// TIA Portal V17 export
// export: Created 2025-03-07T09:23:56.1617823Z, ExportSetting WithDefaults, DisplayName Totally Integrated Automation Portal, DisplayVersion V17 Update 8, DisplayName TIA Portal Openness, DisplayVersion V17 Update 8, DisplayName TIA Portal Version Control Interface, DisplayVersion V17, DisplayName SINAMICS Startdrive Advanced, DisplayVersion V17 SP2, DisplayName SINAMICS Startdrive G110M, G120, G120C, G120D, G120P, G115D, DisplayVersion V17 SP2, DisplayName SINAMICS Startdrive G130, G150, S120, S150, SINAMICS MV, S210, DisplayVersion V17 SP2, DisplayName STEP 7 Professional, DisplayVersion V17 Update 8, DisplayName SINUMERIK ONE STEP 7 Toolbox, DisplayVersion V17 Update 12, DisplayName SINUMERIK 840D sl STEP 7 Toolbox, DisplayVersion V17 Update 12, DisplayName STEP 7 Safety, DisplayVersion V17 Update 6, DisplayName WinCC Advanced, DisplayVersion V17 Update 8
FUNCTION "FC21200_POWDER_FLOW_SENSOR_MEDICOAT" : Void   // FC21200, LAD
{ S7_Optimized_Access := 'TRUE' }
VERSION : 0.1
// stored: AutoNumber false, IsIECCheckEnabled false, SetENOAutomatically false, UDAEnableTagReadback false
BEGIN

REGION Network 1: /////_UNIT_01_/////
END_REGION

REGION Network 2: OERLIKON 1 LINE 1 OUTPUT MEDICOAT
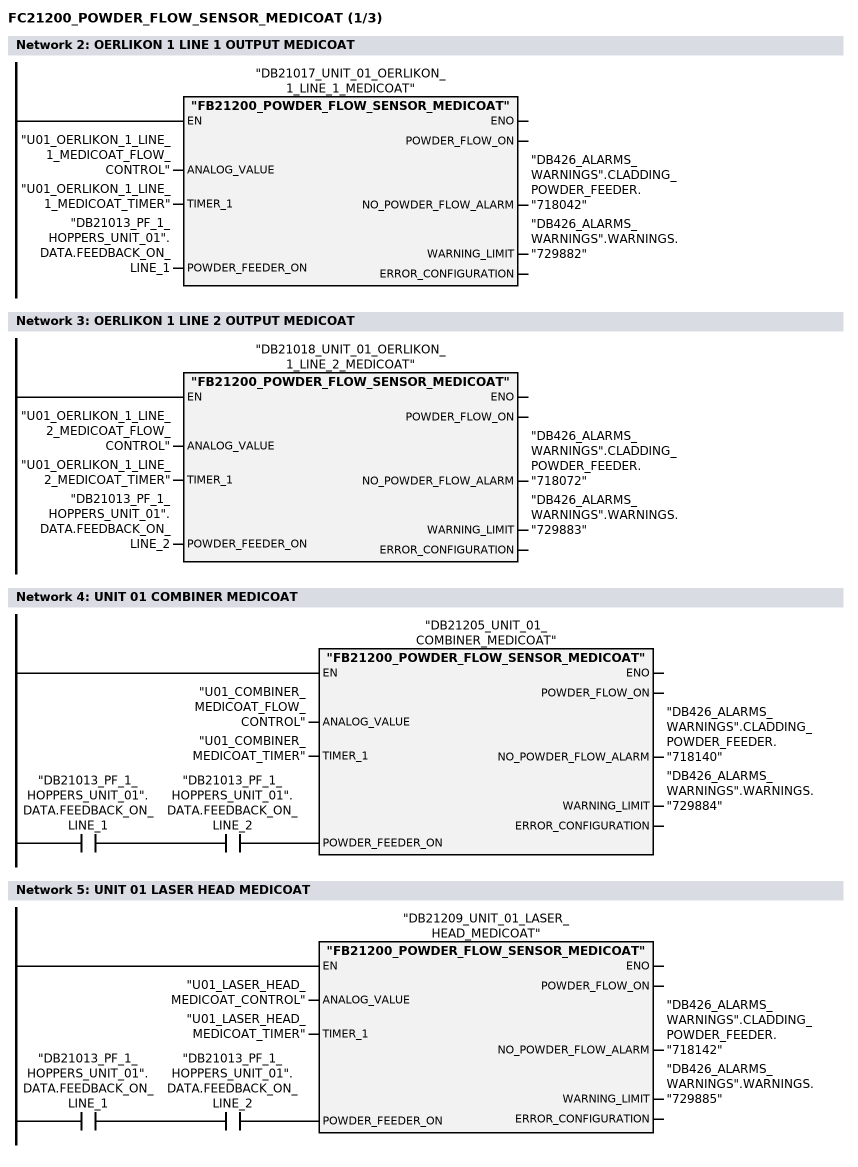
   RUNG wire#powerrail
      "DB21017_UNIT_01_OERLIKON_1_LINE_1_MEDICOAT"(ANALOG_VALUE := "U01_OERLIKON_1_LINE_1_MEDICOAT_FLOW_CONTROL", TIMER_1 := "U01_OERLIKON_1_LINE_1_MEDICOAT_TIMER", POWDER_FEEDER_ON := "DB21013_PF_1_HOPPERS_UNIT_01".DATA.FEEDBACK_ON_LINE_1, POWDER_FLOW_ON =>, NO_POWDER_FLOW_ALARM => "DB426_ALARMS_WARNINGS".CLADDING_POWDER_FEEDER."718042", WARNING_LIMIT => "DB426_ALARMS_WARNINGS".WARNINGS."729882", ERROR_CONFIGURATION =>)
   END_RUNG
   // the same network as SCL:
   "DB21017_UNIT_01_OERLIKON_1_LINE_1_MEDICOAT"(ANALOG_VALUE := "U01_OERLIKON_1_LINE_1_MEDICOAT_FLOW_CONTROL",   // "FB21200_POWDER_FLOW_SENSOR_MEDICOAT"
                           TIMER_1 := "U01_OERLIKON_1_LINE_1_MEDICOAT_TIMER",
                           POWDER_FEEDER_ON := "DB21013_PF_1_HOPPERS_UNIT_01".DATA.FEEDBACK_ON_LINE_1,
                           NO_POWDER_FLOW_ALARM => "DB426_ALARMS_WARNINGS".CLADDING_POWDER_FEEDER."718042",
                           WARNING_LIMIT => "DB426_ALARMS_WARNINGS".WARNINGS."729882");
END_REGION

REGION Network 3: OERLIKON 1 LINE 2 OUTPUT MEDICOAT
   RUNG wire#powerrail
      "DB21018_UNIT_01_OERLIKON_1_LINE_2_MEDICOAT"(ANALOG_VALUE := "U01_OERLIKON_1_LINE_2_MEDICOAT_FLOW_CONTROL", TIMER_1 := "U01_OERLIKON_1_LINE_2_MEDICOAT_TIMER", POWDER_FEEDER_ON := "DB21013_PF_1_HOPPERS_UNIT_01".DATA.FEEDBACK_ON_LINE_2, POWDER_FLOW_ON =>, NO_POWDER_FLOW_ALARM => "DB426_ALARMS_WARNINGS".CLADDING_POWDER_FEEDER."718072", WARNING_LIMIT => "DB426_ALARMS_WARNINGS".WARNINGS."729883", ERROR_CONFIGURATION =>)
   END_RUNG
   // the same network as SCL:
   "DB21018_UNIT_01_OERLIKON_1_LINE_2_MEDICOAT"(ANALOG_VALUE := "U01_OERLIKON_1_LINE_2_MEDICOAT_FLOW_CONTROL",   // "FB21200_POWDER_FLOW_SENSOR_MEDICOAT"
                           TIMER_1 := "U01_OERLIKON_1_LINE_2_MEDICOAT_TIMER",
                           POWDER_FEEDER_ON := "DB21013_PF_1_HOPPERS_UNIT_01".DATA.FEEDBACK_ON_LINE_2,
                           NO_POWDER_FLOW_ALARM => "DB426_ALARMS_WARNINGS".CLADDING_POWDER_FEEDER."718072",
                           WARNING_LIMIT => "DB426_ALARMS_WARNINGS".WARNINGS."729883");
END_REGION

REGION Network 4: UNIT 01 COMBINER MEDICOAT
   RUNG wire#powerrail
      "DB21205_UNIT_01_COMBINER_MEDICOAT"(POWDER_FEEDER_ON := wire#w1, ANALOG_VALUE := "U01_COMBINER_MEDICOAT_FLOW_CONTROL", TIMER_1 := "U01_COMBINER_MEDICOAT_TIMER", POWDER_FLOW_ON =>, NO_POWDER_FLOW_ALARM => "DB426_ALARMS_WARNINGS".CLADDING_POWDER_FEEDER."718140", WARNING_LIMIT => "DB426_ALARMS_WARNINGS".WARNINGS."729884", ERROR_CONFIGURATION =>)
   END_RUNG
   RUNG wire#powerrail
      Contact( "DB21013_PF_1_HOPPERS_UNIT_01".DATA.FEEDBACK_ON_LINE_1 )
      Contact( "DB21013_PF_1_HOPPERS_UNIT_01".DATA.FEEDBACK_ON_LINE_2 )
   END_RUNG wire#w1
   // the same network as SCL:
   "DB21205_UNIT_01_COMBINER_MEDICOAT"(ANALOG_VALUE := "U01_COMBINER_MEDICOAT_FLOW_CONTROL",   // "FB21200_POWDER_FLOW_SENSOR_MEDICOAT"
                           TIMER_1 := "U01_COMBINER_MEDICOAT_TIMER",
                           POWDER_FEEDER_ON := "DB21013_PF_1_HOPPERS_UNIT_01".DATA.FEEDBACK_ON_LINE_1 AND "DB21013_PF_1_HOPPERS_UNIT_01".DATA.FEEDBACK_ON_LINE_2,
                           NO_POWDER_FLOW_ALARM => "DB426_ALARMS_WARNINGS".CLADDING_POWDER_FEEDER."718140",
                           WARNING_LIMIT => "DB426_ALARMS_WARNINGS".WARNINGS."729884");
END_REGION

REGION Network 5: UNIT 01 LASER HEAD MEDICOAT
   RUNG wire#powerrail
      "DB21209_UNIT_01_LASER_HEAD_MEDICOAT"(POWDER_FEEDER_ON := wire#w1, ANALOG_VALUE := "U01_LASER_HEAD_MEDICOAT_CONTROL", TIMER_1 := "U01_LASER_HEAD_MEDICOAT_TIMER", POWDER_FLOW_ON =>, NO_POWDER_FLOW_ALARM => "DB426_ALARMS_WARNINGS".CLADDING_POWDER_FEEDER."718142", WARNING_LIMIT => "DB426_ALARMS_WARNINGS".WARNINGS."729885", ERROR_CONFIGURATION =>)
   END_RUNG
   RUNG wire#powerrail
      Contact( "DB21013_PF_1_HOPPERS_UNIT_01".DATA.FEEDBACK_ON_LINE_1 )
      Contact( "DB21013_PF_1_HOPPERS_UNIT_01".DATA.FEEDBACK_ON_LINE_2 )
   END_RUNG wire#w1
   // the same network as SCL:
   "DB21209_UNIT_01_LASER_HEAD_MEDICOAT"(ANALOG_VALUE := "U01_LASER_HEAD_MEDICOAT_CONTROL",   // "FB21200_POWDER_FLOW_SENSOR_MEDICOAT"
                           TIMER_1 := "U01_LASER_HEAD_MEDICOAT_TIMER",
                           POWDER_FEEDER_ON := "DB21013_PF_1_HOPPERS_UNIT_01".DATA.FEEDBACK_ON_LINE_1 AND "DB21013_PF_1_HOPPERS_UNIT_01".DATA.FEEDBACK_ON_LINE_2,
                           NO_POWDER_FLOW_ALARM => "DB426_ALARMS_WARNINGS".CLADDING_POWDER_FEEDER."718142",
                           WARNING_LIMIT => "DB426_ALARMS_WARNINGS".WARNINGS."729885");
END_REGION

REGION Network 6: /////_UNIT_02_/////
END_REGION

REGION Network 7: UNIT 02 OERLIKON 1 LINE 1 OUTPUT MEDICOAT
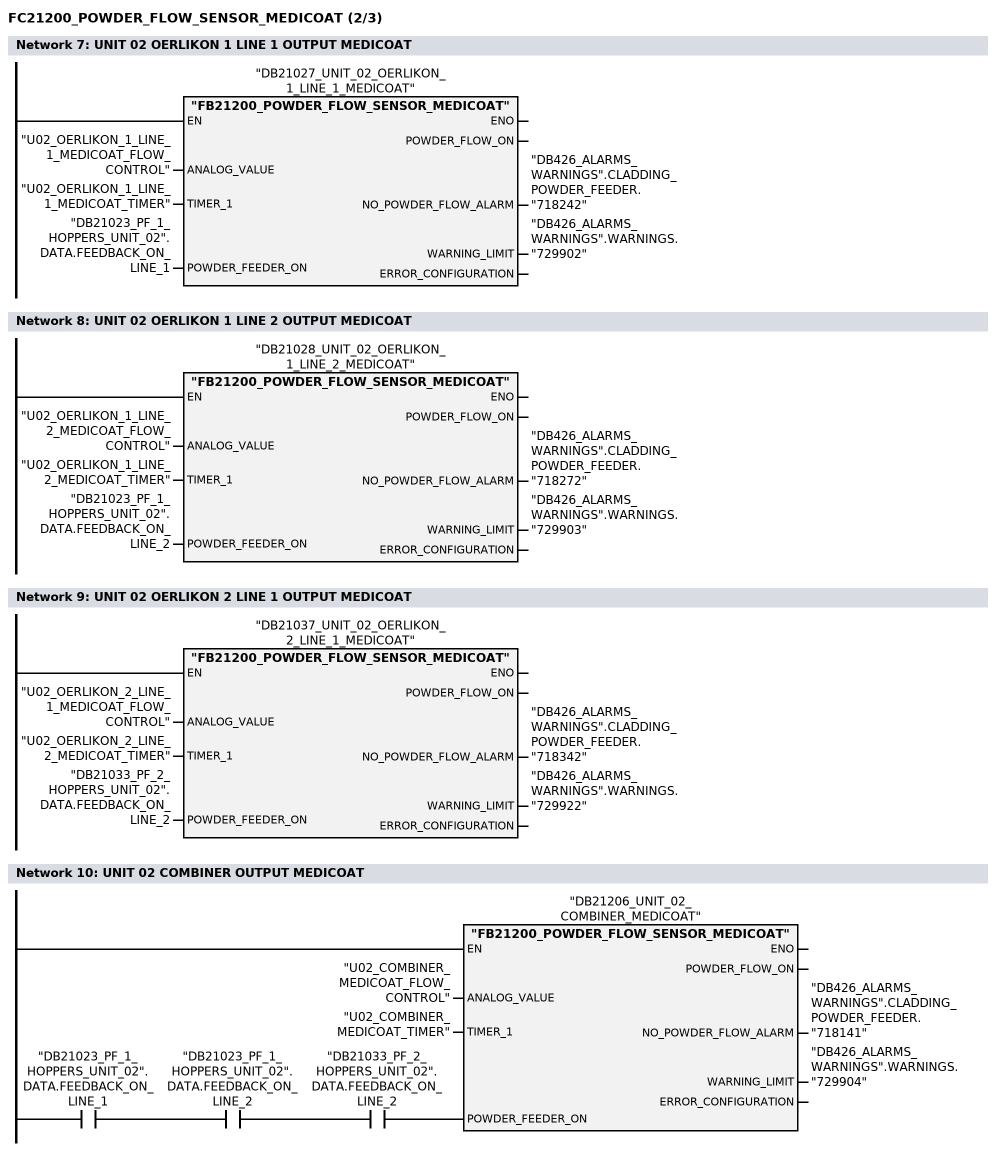
   RUNG wire#powerrail
      "DB21027_UNIT_02_OERLIKON_1_LINE_1_MEDICOAT"(ANALOG_VALUE := "U02_OERLIKON_1_LINE_1_MEDICOAT_FLOW_CONTROL", TIMER_1 := "U02_OERLIKON_1_LINE_1_MEDICOAT_TIMER", POWDER_FEEDER_ON := "DB21023_PF_1_HOPPERS_UNIT_02".DATA.FEEDBACK_ON_LINE_1, POWDER_FLOW_ON =>, NO_POWDER_FLOW_ALARM => "DB426_ALARMS_WARNINGS".CLADDING_POWDER_FEEDER."718242", WARNING_LIMIT => "DB426_ALARMS_WARNINGS".WARNINGS."729902", ERROR_CONFIGURATION =>)
   END_RUNG
   // the same network as SCL:
   "DB21027_UNIT_02_OERLIKON_1_LINE_1_MEDICOAT"(ANALOG_VALUE := "U02_OERLIKON_1_LINE_1_MEDICOAT_FLOW_CONTROL",   // "FB21200_POWDER_FLOW_SENSOR_MEDICOAT"
                           TIMER_1 := "U02_OERLIKON_1_LINE_1_MEDICOAT_TIMER",
                           POWDER_FEEDER_ON := "DB21023_PF_1_HOPPERS_UNIT_02".DATA.FEEDBACK_ON_LINE_1,
                           NO_POWDER_FLOW_ALARM => "DB426_ALARMS_WARNINGS".CLADDING_POWDER_FEEDER."718242",
                           WARNING_LIMIT => "DB426_ALARMS_WARNINGS".WARNINGS."729902");
END_REGION

REGION Network 8: UNIT 02 OERLIKON 1 LINE 2 OUTPUT MEDICOAT
   RUNG wire#powerrail
      "DB21028_UNIT_02_OERLIKON_1_LINE_2_MEDICOAT"(ANALOG_VALUE := "U02_OERLIKON_1_LINE_2_MEDICOAT_FLOW_CONTROL", TIMER_1 := "U02_OERLIKON_1_LINE_2_MEDICOAT_TIMER", POWDER_FEEDER_ON := "DB21023_PF_1_HOPPERS_UNIT_02".DATA.FEEDBACK_ON_LINE_2, POWDER_FLOW_ON =>, NO_POWDER_FLOW_ALARM => "DB426_ALARMS_WARNINGS".CLADDING_POWDER_FEEDER."718272", WARNING_LIMIT => "DB426_ALARMS_WARNINGS".WARNINGS."729903", ERROR_CONFIGURATION =>)
   END_RUNG
   // the same network as SCL:
   "DB21028_UNIT_02_OERLIKON_1_LINE_2_MEDICOAT"(ANALOG_VALUE := "U02_OERLIKON_1_LINE_2_MEDICOAT_FLOW_CONTROL",   // "FB21200_POWDER_FLOW_SENSOR_MEDICOAT"
                           TIMER_1 := "U02_OERLIKON_1_LINE_2_MEDICOAT_TIMER",
                           POWDER_FEEDER_ON := "DB21023_PF_1_HOPPERS_UNIT_02".DATA.FEEDBACK_ON_LINE_2,
                           NO_POWDER_FLOW_ALARM => "DB426_ALARMS_WARNINGS".CLADDING_POWDER_FEEDER."718272",
                           WARNING_LIMIT => "DB426_ALARMS_WARNINGS".WARNINGS."729903");
END_REGION

REGION Network 9: UNIT 02 OERLIKON 2 LINE 1 OUTPUT MEDICOAT
   RUNG wire#powerrail
      "DB21037_UNIT_02_OERLIKON_2_LINE_1_MEDICOAT"(ANALOG_VALUE := "U02_OERLIKON_2_LINE_1_MEDICOAT_FLOW_CONTROL", TIMER_1 := "U02_OERLIKON_2_LINE_2_MEDICOAT_TIMER", POWDER_FEEDER_ON := "DB21033_PF_2_HOPPERS_UNIT_02".DATA.FEEDBACK_ON_LINE_2, POWDER_FLOW_ON =>, NO_POWDER_FLOW_ALARM => "DB426_ALARMS_WARNINGS".CLADDING_POWDER_FEEDER."718342", WARNING_LIMIT => "DB426_ALARMS_WARNINGS".WARNINGS."729922", ERROR_CONFIGURATION =>)
   END_RUNG
   // the same network as SCL:
   "DB21037_UNIT_02_OERLIKON_2_LINE_1_MEDICOAT"(ANALOG_VALUE := "U02_OERLIKON_2_LINE_1_MEDICOAT_FLOW_CONTROL",   // "FB21200_POWDER_FLOW_SENSOR_MEDICOAT"
                           TIMER_1 := "U02_OERLIKON_2_LINE_2_MEDICOAT_TIMER",
                           POWDER_FEEDER_ON := "DB21033_PF_2_HOPPERS_UNIT_02".DATA.FEEDBACK_ON_LINE_2,
                           NO_POWDER_FLOW_ALARM => "DB426_ALARMS_WARNINGS".CLADDING_POWDER_FEEDER."718342",
                           WARNING_LIMIT => "DB426_ALARMS_WARNINGS".WARNINGS."729922");
END_REGION

REGION Network 10: UNIT 02 COMBINER OUTPUT MEDICOAT
   RUNG wire#powerrail
      "DB21206_UNIT_02_COMBINER_MEDICOAT"(POWDER_FEEDER_ON := wire#w1, ANALOG_VALUE := "U02_COMBINER_MEDICOAT_FLOW_CONTROL", TIMER_1 := "U02_COMBINER_MEDICOAT_TIMER", POWDER_FLOW_ON =>, NO_POWDER_FLOW_ALARM => "DB426_ALARMS_WARNINGS".CLADDING_POWDER_FEEDER."718141", WARNING_LIMIT => "DB426_ALARMS_WARNINGS".WARNINGS."729904", ERROR_CONFIGURATION =>)
   END_RUNG
   RUNG wire#powerrail
      Contact( "DB21023_PF_1_HOPPERS_UNIT_02".DATA.FEEDBACK_ON_LINE_1 )
      Contact( "DB21023_PF_1_HOPPERS_UNIT_02".DATA.FEEDBACK_ON_LINE_2 )
      Contact( "DB21033_PF_2_HOPPERS_UNIT_02".DATA.FEEDBACK_ON_LINE_2 )
   END_RUNG wire#w1
   // the same network as SCL:
   "DB21206_UNIT_02_COMBINER_MEDICOAT"(ANALOG_VALUE := "U02_COMBINER_MEDICOAT_FLOW_CONTROL",   // "FB21200_POWDER_FLOW_SENSOR_MEDICOAT"
                           TIMER_1 := "U02_COMBINER_MEDICOAT_TIMER",
                           POWDER_FEEDER_ON := "DB21023_PF_1_HOPPERS_UNIT_02".DATA.FEEDBACK_ON_LINE_1 AND "DB21023_PF_1_HOPPERS_UNIT_02".DATA.FEEDBACK_ON_LINE_2 AND "DB21033_PF_2_HOPPERS_UNIT_02".DATA.FEEDBACK_ON_LINE_2,
                           NO_POWDER_FLOW_ALARM => "DB426_ALARMS_WARNINGS".CLADDING_POWDER_FEEDER."718141",
                           WARNING_LIMIT => "DB426_ALARMS_WARNINGS".WARNINGS."729904");
END_REGION

REGION Network 11: UNIT 02 LASER HEAD OUTPUT MEDICOAT
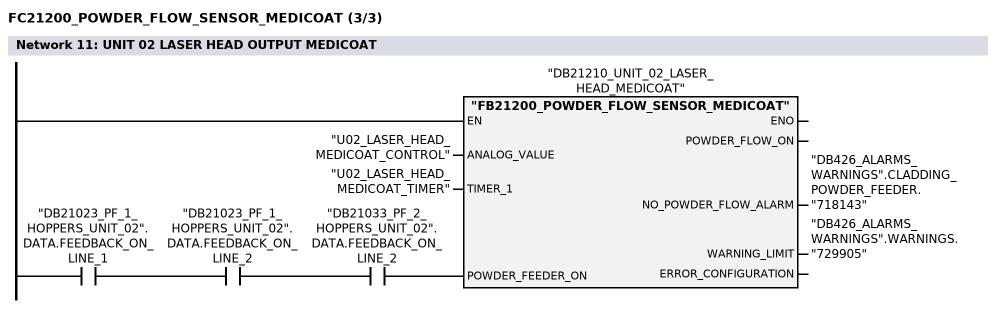
   RUNG wire#powerrail
      "DB21210_UNIT_02_LASER_HEAD_MEDICOAT"(POWDER_FEEDER_ON := wire#w1, ANALOG_VALUE := "U02_LASER_HEAD_MEDICOAT_CONTROL", TIMER_1 := "U02_LASER_HEAD_MEDICOAT_TIMER", POWDER_FLOW_ON =>, NO_POWDER_FLOW_ALARM => "DB426_ALARMS_WARNINGS".CLADDING_POWDER_FEEDER."718143", WARNING_LIMIT => "DB426_ALARMS_WARNINGS".WARNINGS."729905", ERROR_CONFIGURATION =>)
   END_RUNG
   RUNG wire#powerrail
      Contact( "DB21023_PF_1_HOPPERS_UNIT_02".DATA.FEEDBACK_ON_LINE_1 )
      Contact( "DB21023_PF_1_HOPPERS_UNIT_02".DATA.FEEDBACK_ON_LINE_2 )
      Contact( "DB21033_PF_2_HOPPERS_UNIT_02".DATA.FEEDBACK_ON_LINE_2 )
   END_RUNG wire#w1
   // the same network as SCL:
   "DB21210_UNIT_02_LASER_HEAD_MEDICOAT"(ANALOG_VALUE := "U02_LASER_HEAD_MEDICOAT_CONTROL",   // "FB21200_POWDER_FLOW_SENSOR_MEDICOAT"
                           TIMER_1 := "U02_LASER_HEAD_MEDICOAT_TIMER",
                           POWDER_FEEDER_ON := "DB21023_PF_1_HOPPERS_UNIT_02".DATA.FEEDBACK_ON_LINE_1 AND "DB21023_PF_1_HOPPERS_UNIT_02".DATA.FEEDBACK_ON_LINE_2 AND "DB21033_PF_2_HOPPERS_UNIT_02".DATA.FEEDBACK_ON_LINE_2,
                           NO_POWDER_FLOW_ALARM => "DB426_ALARMS_WARNINGS".CLADDING_POWDER_FEEDER."718143",
                           WARNING_LIMIT => "DB426_ALARMS_WARNINGS".WARNINGS."729905");
END_REGION
END_FUNCTION
